ABB RobotStudio station: FinalSystem_Mark5.rspag

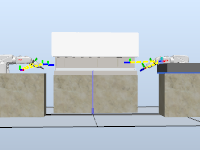
--- station ---
Station FinalSystem_Mark5 (saved by RobotStudio 20.1.8982.0)
Controller Brazo_Izquierdo, task T_ROB1: task frame (RAPID world) sits at (381.13, 1073.42, 0) mm, rotated rx 0 ry 0.08 rz -90.05 deg in the station
Controller Brazo_Derecho, task T_ROB1: task frame (RAPID world) sits at (383.2, -1129.52, 0) mm, rotated rx 0 ry 0 rz 90 deg in the station
Controller Brazo_Derecho
  mechanical unit ROB_1: Brazo_Derecho, 6 joints, base frame (0, 0, 0) mm
Controller Brazo_Izquierdo
  mechanical unit ROB_1: Brazo_Izquierdo, 6 joints, base frame (0, 0, 0) mm
Layout (positions relative to the parent item):
  - Drunk machine [part] at (-616.69, -0.57, 747.91) mm, rotated rx 90.16 ry 0 rz 90.05 deg
  - rack [part] at (-166.71, -1080.65, 472.06) mm
  - ASS Nastro 80 [graphiccomponentgroup] at (220.02, -32.24, 435.23) mm, rotated rx -89.85 ry 0 rz 90.13 deg
    - Spalla ant tappeto-1 [part] at (3.95, -82.87, -3) mm
    - Tappeto L500 d80-1 [part] at (-9.66, -82.87, -105) mm
    - Spalla post tappeto 80-2 [part] at (3.95, -82.87, -207) mm
    - Traversa supporto piano di lavoro Nastro 80-1 [part] at (3.95, -77.67, -105) mm
    - Traversa supporto piano di lavoro Nastro 80-2 [part] at (363.95, -77.67, -105) mm
    - Traversa supporto piano di lavoro Nastro 80-3 [part] at (243.95, -77.67, -105) mm
    - Traversa supporto piano di lavoro Nastro 80-4 [part] at (123.95, -77.67, -105) mm
    - Traversa supporto piano di lavoro Nastro 80-5 [part] at (-116.05, -77.67, -105) mm
    - Ass rullo passivo Nastro 80-1 [graphiccomponentgroup] at (-483.55, -82.94, -125) mm, rotated rx 0 ry 0 rz 115.98 deg
      - Albero rullo passivo 80-1 [part] at (-0.06, -0.28, -82) mm
      - Rullo passivo Nastro 80-1 [part] at (-0.06, -0.28, 20) mm, rotated rx 0 ry 0 rz 44.34 deg
      - Cuscinetto 6205-2RS1-2 [part] at (-0.06, -0.28, 121) mm, rotated rx 0 ry 90 rz -50.21 deg
      - Cuscinetto 6205-2RS1-3 [part] at (-0.06, -0.28, -75) mm, rotated rx 0 ry 90 rz -77.93 deg
    - Traversa supporto piano di lavoro Nastro 80-6 [part] at (-236.05, -77.67, -105) mm
    - Traversa supporto piano di lavoro Nastro 80-7 [part] at (-356.05, -77.67, -105) mm
    - Testa spalla front Nastro 80-1 [part] at (-483.27, -82.87, 0) mm
    - Testa spalla post Nastro 80-1 [part] at (-483.27, -82.87, -210) mm
  - Brazo_Izquierdo [mechanism, from Robots\IRB120_3_58_G_01.rslib] at (381.13, 1073.42, 0) mm, rotated rx 0 ry 0.08 rz -90.05 deg; joint values [0, 0, 0, 0, 0.5236, 1.5708] (rad or m)
  - Smart_Gripper_Servo_Fingers [mechanism, from Libraries\Smart_Gripper2.rslib] at (383.22, -765.16, 594) mm, rotated rx 120 ry 0 rz 180 deg; joint values [0.025] (rad or m)
  - Brazo_Derecho [mechanism, from Robots\IRB120_3_58_G_01.rslib] at (383.2, -1129.52, 0) mm, rotated rx 0 ry 0 rz 90 deg; joint values [0, 0, 0, 0, 0.5236, 1.5708] (rad or m)
  - Smart_Gripper_Servo_Fingers_2 [mechanism, from Tools\ABB_Smart_Gripper_Servo_Fingers.rslib] at (380.83, 708.25, 593.49) mm, rotated rx 120.08 ry 0 rz -0.05 deg; joint values [0.0241] (rad or m)
  - Base [part] at (176.64, -543.05, 0) mm
  - Vaso [part] at (55.85, -802.14, 590.8) mm
  - Positioner [smart component, from Components\Positioner.rslib]
      properties: Object=Vaso; Position=[0.055849 -0.80214 0.5908]; Orientation=[0 0 0]; Reference=Global; ReferenceObject=(none)
  - Sensor_Final [smart component, from Components\PlaneSensor.rslib] at (317.79, 437.34, 555.44) mm, rotated rx 90 ry 0 rz 0 deg
      properties: Origin=[0 0 0]; Axis1=[0.1 0 0]; Axis2=[0 0.1 0]; SensedPart=(none)
    - _sensorPart_ [part, from Components\PlaneSensor.rslib]
  - SimulationEvents [smart component, from Components\SimulationEvents.rslib]
  - LogicSRLatch [smart component, from Components\LogicSRLatch.rslib]
  - LinearMover_I-H [smart component, from Components\LinearMover.rslib]
      properties: Object=Vaso; Direction=[0 0.1 0]; Speed=0.06; Reference=Global; ReferenceObject=(none)
  - Detacher [smart component, from Components\Detacher.rslib]
      properties: Child=Vaso; KeepPosition=true
  - Sensor_Hielos [smart component, from Components\PlaneSensor.rslib] at (291.31, -320.38, 553.19) mm, rotated rx 90 ry 0 rz 0 deg
      properties: Origin=[0 0 0]; Axis1=[0.1 0 0]; Axis2=[0 0.1 0]; SensedPart=(none)
    - _sensorPart_ [part, from Components\PlaneSensor.rslib]
  - Attacher_2 [smart component, from Components\Attacher.rslib]
      properties: Parent=Smart_Gripper_Servo_Fingers_2; Flange=0; Child=Vaso; Mount=false; Offset=[0 0 0]; Orientation=[0 0 0]
  - Pieza_8 [part] at (-304.73, -1255.96, -1.15) mm
  - Pieza_9 [part] at (-221.9, 531.96, -0.59) mm
  - Attacher_3 [smart component, from Components\Attacher.rslib]
      properties: Parent=Smart_Gripper_Servo_Fingers; Flange=0; Child=Vaso; Mount=false; Offset=[0 0 0]; Orientation=[0 0 0]
  - Detacher_2 [smart component, from Components\Detacher.rslib]
      properties: Child=Vaso; KeepPosition=true
  - LinearMover_H-A [smart component, from Components\LinearMover.rslib]
      properties: Object=Vaso; Direction=[0 0.1 0]; Speed=0.06; Reference=Global; ReferenceObject=(none)
  - LogicSRLatch_2 [smart component, from Components\LogicSRLatch.rslib]
  - Sensor_Tequila [smart component, from Components\PlaneSensor.rslib] at (290.86, -66.85, 550.9) mm, rotated rx 90 ry 0 rz 0 deg
      properties: Origin=[0 0 0]; Axis1=[0.1 0 0]; Axis2=[0 0.1 0]; SensedPart=(none)
    - _sensorPart_ [part, from Components\PlaneSensor.rslib]
  - LinearMover_A-M [smart component, from Components\LinearMover.rslib]
      properties: Object=Vaso; Direction=[0 0.1 0]; Speed=0.06; Reference=Global; ReferenceObject=(none)
  - LogicSRLatch_3 [smart component, from Components\LogicSRLatch.rslib]
  - Sensor_Toronja [smart component, from Components\PlaneSensor.rslib] at (305.49, 235.87, 549.38) mm, rotated rx 90 ry 0 rz 0 deg
      properties: Origin=[0 0 0]; Axis1=[0.1 0 0]; Axis2=[0 0.1 0]; SensedPart=(none)
    - _sensorPart_ [part, from Components\PlaneSensor.rslib]
  - LogicSRLatch_4 [smart component, from Components\LogicSRLatch.rslib]
  - LinearMover_M-F [smart component, from Components\LinearMover.rslib]
      properties: Object=Vaso; Direction=[0 0.1 0]; Speed=0.06; Reference=Global; ReferenceObject=(none)
  - Sensor_Coca [smart component, from Components\PlaneSensor.rslib] at (296.45, 334.57, 549.82) mm, rotated rx 90 ry 0 rz 0 deg
      properties: Origin=[0 0 0]; Axis1=[0.1 0 0]; Axis2=[0 0.1 0]; SensedPart=(none)
    - _sensorPart_ [part, from Components\PlaneSensor.rslib]
  - LogicSRLatch_5 [smart component, from Components\LogicSRLatch.rslib]
  - Sensor_Sprite [smart component, from Components\PlaneSensor.rslib] at (304.78, 430.43, 554.72) mm, rotated rx 90 ry 0 rz 0 deg
      properties: Origin=[0 0 0]; Axis1=[0.1 0 0]; Axis2=[0 0.1 0]; SensedPart=(none)
    - _sensorPart_ [part, from Components\PlaneSensor.rslib]
  - LogicSRLatch_6 [smart component, from Components\LogicSRLatch.rslib]
  - LogicSRLatch_7 [smart component, from Components\LogicSRLatch.rslib]
  - Sensor_Vodka [smart component, from Components\PlaneSensor.rslib] at (307.92, 135.66, 549.24) mm, rotated rx 90 ry 0 rz 0 deg
      properties: Origin=[0 0 0]; Axis1=[0.1 0 0]; Axis2=[0 0.1 0]; SensedPart=(none)
    - _sensorPart_ [part, from Components\PlaneSensor.rslib]
Attachment: Smart_Gripper_Servo_Fingers is attached to Brazo_Derecho / Link6
Attachment: Smart_Gripper_Servo_Fingers_2 is attached to Brazo_Izquierdo / Link6
Station signals: DI Posicionador
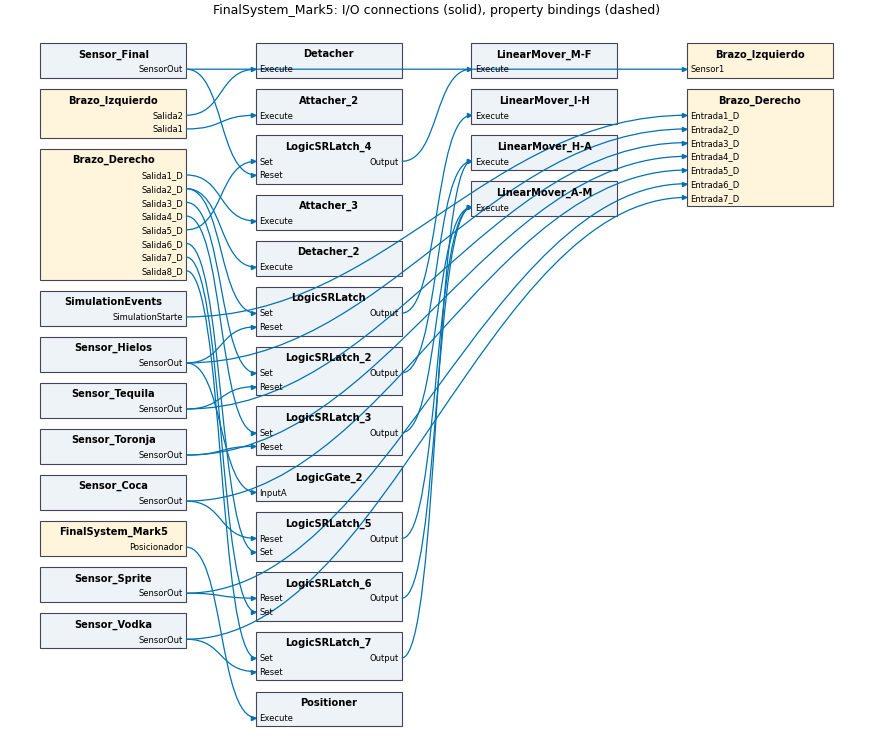
Station logic (signal -> signal, property => property):
  Sensor_Final.SensorOut -> Brazo_Izquierdo.Sensor1
  LogicSRLatch.Output -> LinearMover_I-H.Execute
  Brazo_Izquierdo.Salida2 -> Detacher.Execute
  Brazo_Izquierdo.Salida1 -> Attacher_2.Execute
  Brazo_Derecho.Salida1_D -> Attacher_3.Execute
  Brazo_Derecho.Salida2_D -> Detacher_2.Execute
  SimulationEvents.SimulationStarted -> Brazo_Derecho.Entrada1_D
  Sensor_Hielos.SensorOut -> LogicGate_2.InputA
  Brazo_Derecho.Salida2_D -> LogicSRLatch.Set
  Sensor_Hielos.SensorOut -> LogicSRLatch.Reset
  Brazo_Derecho.Salida3_D -> LogicSRLatch_2.Set
  LogicSRLatch_2.Output -> LinearMover_H-A.Execute
  Sensor_Hielos.SensorOut -> Brazo_Derecho.Entrada2_D
  Brazo_Derecho.Salida4_D -> LogicSRLatch_3.Set
  LogicSRLatch_3.Output -> LinearMover_A-M.Execute
  Sensor_Tequila.SensorOut -> Brazo_Derecho.Entrada3_D
  Sensor_Tequila.SensorOut -> LogicSRLatch_2.Reset
  Sensor_Toronja.SensorOut -> Brazo_Derecho.Entrada4_D
  Sensor_Toronja.SensorOut -> LogicSRLatch_3.Reset
  Brazo_Derecho.Salida5_D -> LogicSRLatch_4.Set
  Sensor_Final.SensorOut -> LogicSRLatch_4.Reset
  LogicSRLatch_4.Output -> LinearMover_M-F.Execute
  Sensor_Coca.SensorOut -> Brazo_Derecho.Entrada5_D
  FinalSystem_Mark5.Posicionador -> Positioner.Execute
  LogicSRLatch_5.Output -> LinearMover_A-M.Execute
  Sensor_Coca.SensorOut -> LogicSRLatch_5.Reset
  Brazo_Derecho.Salida6_D -> LogicSRLatch_5.Set
  Sensor_Sprite.SensorOut -> Brazo_Derecho.Entrada6_D
  Sensor_Sprite.SensorOut -> LogicSRLatch_6.Reset
  Brazo_Derecho.Salida7_D -> LogicSRLatch_6.Set
  LogicSRLatch_6.Output -> LinearMover_A-M.Execute
  Sensor_Vodka.SensorOut -> Brazo_Derecho.Entrada7_D
  Brazo_Derecho.Salida8_D -> LogicSRLatch_7.Set
  Sensor_Vodka.SensorOut -> LogicSRLatch_7.Reset
  LogicSRLatch_7.Output -> LinearMover_H-A.Execute

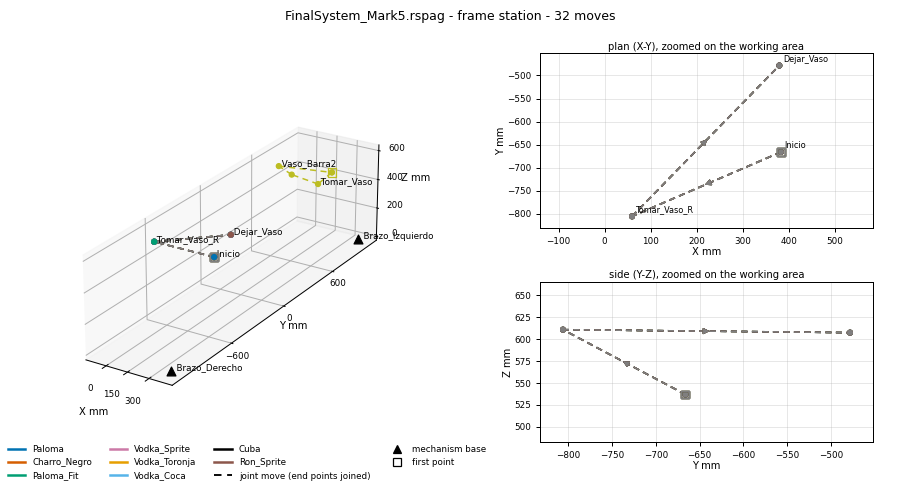
[picture p0: tool path of FinalSystem_Mark5.rspag in frame station, 32 of 32 moves have a stored position in this frame; points joined in program order, loops and branches not executed]
--- Backups/Brazo_Derecho/RAPID/TASK1/PROGMOD/CalibData.mod ---
MODULE CalibData
    PERS tooldata Servo:=[TRUE,[[0,0,114.2],[1,0,0,0]],[0.215,[8.7,12.3,49.2],[1,0,0,0],0.00021,0.00024,0.00009]];
ENDMODULE

--- Backups/Brazo_Derecho/RAPID/TASK1/PROGMOD/Module1.mod ---
MODULE Module1
    CONST robtarget Home:=[[463.253923278,0,536.899988039],[0.353553368,0.612372449,0.612372449,0.353553368],[0,-1,1,0],[9E+09,9E+09,9E+09,9E+09,9E+09,9E+09]];
    CONST robtarget AbovePickPosition:=[[323.968763837,312.895755919,276.594],[0.707106781,-0.707106781,-0.000020041,0.000020041],[0,0,0,0],[9E+09,9E+09,9E+09,9E+09,9E+09,9E+09]];
    CONST robtarget PickPosition:=[[323.968763837,312.895755919,156.594],[0.707106781,-0.707106781,-0.000020041,0.000020041],[0,0,0,0],[9E+09,9E+09,9E+09,9E+09,9E+09,9E+09]];
    CONST robtarget Inicio:=[[463.253923278,0,536.899988039],[0.353553368,0.612372449,0.612372449,0.353553368],[0,-1,1,0],[9E+09,9E+09,9E+09,9E+09,9E+09,9E+09]];
    CONST robtarget Tomar_Vaso_R:=[[323.459576854,323.459552433,610.906782794],[0.265834211,0.275279486,0.664583392,0.641780564],[0,0,1,0],[9E+09,9E+09,9E+09,9E+09,9E+09,9E+09]];
    CONST robtarget Dejar_Vaso:=[[651.164684644,3.54793506,607.492960443],[0.494318369,0.503022234,0.50566295,0.496913436],[0,-1,1,0],[9E+09,9E+09,9E+09,9E+09,9E+09,9E+09]];
   PROC main()
!        VAR socketdev server_socket;
!        VAR socketdev client_socket;
!        VAR string client_ip;
!        VAR string drinkID;
!        VAR bool loop:=TRUE;


!        SocketCreate server_socket;
!        SocketBind server_socket, "127.0.0.1", 55555;
!        SocketListen server_socket;

        ! Waiting for a connection request
!        SocketAccept server_socket, client_socket\ClientAddress:=client_ip\Time:=WAIT_MAX;

!        WHILE loop DO

!            SocketReceive client_socket \Str := drinkID\Time:=WAIT_MAX;

            !State machine
!            IF drinkID="id" THEN
!                !Mover izquierda
!                TPWrite "Izquierda";
!                Path_10;
!            ENDIF

!            drinkID := "";

            !Send acknowledge
            !SocketSend client_socket \Str := "Hello client with ip-addres " +client_ip;
!        ENDWHILE
!    ERROR
!        RETRY;
!    UNDO
!        SocketClose server_socket;
!        SocketClose client_socket;
        !Paloma;
        !Charro_Negro;
        !Paloma_Fit;
        !Vodka_Sprite;
        !Vodka_Toronja;
        !Vodka_Coca;
        !Cuba;
        !Ron_Sprite;
        Ron_Toronja;
    ENDPROC

    PROC Paloma()
        SetDO Salida1_D,0;
        SetDO Salida2_D,0;
        SetDO Salida3_D,0;
        SetDO Salida4_D,0;
        SetDO Salida5_D,0;
        SetDO Salida6_D,0;
        SetDO Salida7_D,0;
        SetDO Salida8_D,0;
        SetDO Salida9_D,0;

        !Movimiento Inicial Secuencia
        WaitDI Entrada1_D,1; !Espera a que se inicie la simulación
        MoveJ Inicio,v100,fine,Servo\WObj:=wobj0;!Mueve el brazo a posicion Inicial
        WaitTime 1;!Espera un segundo
        MoveJ Tomar_Vaso_R,v1000,fine,Servo\WObj:=wobj0;!Mueve el brazo a tomar el vaso
        WaitTime 1;!Espera un segundo
        SetDO Salida1_D,1;!Inicializa la salida1 a 1 para atach el vaso
        WaitTime 1;!Espera un segundo
        MoveJ Dejar_Vaso,v1000,fine,Servo\WObj:=wobj0; !Mueve el brazo y el vaso a la conveyor belt
        WaitTime 1;!Espera un segundo
        SetDO Salida1_D,0;!Inicializa la salida1 a 0 para deatach el vaso

        !Movimiento de Inicio a Sensor Hielos
        SetDO Salida2_D,1;!Inicializa la salida2 a 1 para iniciar LinearMover_I-H
        WaitTime 1;!Espera un segundo
        SetDO Salida2_D,0;!Inicializa la salida2 a 0 para evitar inicializar el LinearMover_I-H de nuevo.
        WaitDI Entrada2_D,1;!Espera a que el sensor hielos se active y para el movimiento.
        WaitTime 3;!Espera tres segundos en servir hielos

        !Movimiento de Sensor Hielos a Sensor A1
        SetDO Salida3_D,1;!Inicializa la salida3 a 1 para iniciar LinearMover_H-A
        WaitTime 1;!Espera un segundo
        SetDO Salida3_D,0;!Inicializa la salida3 a 0 para evitar inicializar el LinearMover_I-H de nuevo.
        WaitDI Entrada3_D,1;
        WaitTime 4;!Espera cuatro segundos en servir alcohol

        !Movimiento de Sensor A1 a Sensor M1
        SetDO Salida4_D,1;!Inicializa la salida4 a 1 para iniciar LinearMover_A-M
        WaitTime 1;!Espera un segundo
        SetDO Salida4_D,0;!Inicializa la salida4 a 0 para evitar inicializar el LinearMover_I-H de nuevo.
        WaitDI Entrada4_D,1;
        WaitTime 7;!Espera siete segundos en servir mixer

        !Movimiento de Sensor M1 a Sensor Final
        SetDO Salida5_D,1; !Inicializa la salida5 a 1 para iniciar LinearMover_M-F
        WaitTime 1;!Espera un segundo
        SetDO Salida5_D,0;!Inicializa la salida4 a 0 para evitar inicializar el LinearMover_I-H de nuevo.
    ENDPROC

    PROC Charro_Negro()
        SetDO Salida1_D,0;
        SetDO Salida2_D,0;
        SetDO Salida3_D,0;
        SetDO Salida4_D,0;
        SetDO Salida5_D,0;
        SetDO Salida6_D,0;
        SetDO Salida7_D,0;
        SetDO Salida8_D,0;
        SetDO Salida9_D,0;

        !Movimiento Inicial Secuencia
        WaitDI Entrada1_D,1; !Espera a que se inicie la simulación
        MoveJ Inicio,v100,fine,Servo\WObj:=wobj0;!Mueve el brazo a posicion Inicial
        WaitTime 1;!Espera un segundo
        MoveJ Tomar_Vaso_R,v1000,fine,Servo\WObj:=wobj0;!Mueve el brazo a tomar el vaso
        WaitTime 1;!Espera un segundo
        SetDO Salida1_D,1;!Inicializa la salida1 a 1 para atach el vaso
        WaitTime 1;!Espera un segundo
        MoveJ Dejar_Vaso,v1000,fine,Servo\WObj:=wobj0; !Mueve el brazo y el vaso a la conveyor belt
        WaitTime 1;!Espera un segundo
        SetDO Salida1_D,0;!Inicializa la salida1 a 0 para deatach el vaso

        !Movimiento de Inicio a Sensor Hielos
        SetDO Salida2_D,1;!Inicializa la salida2 a 1 para iniciar LinearMover_I-H
        WaitTime 1;!Espera un segundo
        SetDO Salida2_D,0;!Inicializa la salida2 a 0 para evitar inicializar el LinearMover_I-H de nuevo.
        WaitDI Entrada2_D,1;!Espera a que el sensor hielos se active y para el movimiento.
        WaitTime 3;!Espera tres segundos en servir hielos

        !Movimiento de Sensor Hielos a Sensor Tequila
        SetDO Salida3_D,1;!Inicializa la salida3 a 1 para iniciar LinearMover_H-A
        WaitTime 1;!Espera un segundo
        SetDO Salida3_D,0;!Inicializa la salida3 a 0 para evitar inicializar el LinearMover_H-A de nuevo.
        WaitDI Entrada3_D,1;
        WaitTime 4;!Espera cuatro segundos en servir alcohol

        !Movimiento de Sensor Tequila a Sensor Coca
        SetDO Salida6_D,1;!Inicializa la salida7 a 1 para iniciar LinearMover_A-M
        WaitTime 1;!Espera un segundo
        SetDO Salida6_D,0;!Inicializa la salida4 a 0 para evitar inicializar el LinearMover_I-H de nuevo.
        WaitDI Entrada5_D,1;
        WaitTime 7;!Espera siete segundos en servir mixer

        !Movimiento de Sensor M1 a Sensor Final
        SetDO Salida5_D,1; !Inicializa la salida5 a 1 para iniciar LinearMover_M-F
        WaitTime 1;!Espera un segundo
        SetDO Salida5_D,0;!Inicializa la salida4 a 0 para evitar inicializar el LinearMover_I-H de nuevo.
    ENDPROC

    PROC Paloma_Fit()
        SetDO Salida1_D,0;
        SetDO Salida2_D,0;
        SetDO Salida3_D,0;
        SetDO Salida4_D,0;
        SetDO Salida5_D,0;
        SetDO Salida6_D,0;
        SetDO Salida7_D,0;
        SetDO Salida8_D,0;
        SetDO Salida9_D,0;

        !Movimiento Inicial Secuencia
        WaitDI Entrada1_D,1; !Espera a que se inicie la simulación
        MoveJ Inicio,v100,fine,Servo\WObj:=wobj0;!Mueve el brazo a posicion Inicial
        WaitTime 1;!Espera un segundo
        MoveJ Tomar_Vaso_R,v1000,fine,Servo\WObj:=wobj0;!Mueve el brazo a tomar el vaso
        WaitTime 1;!Espera un segundo
        SetDO Salida1_D,1;!Inicializa la salida1 a 1 para atach el vaso
        WaitTime 1;!Espera un segundo
        MoveJ Dejar_Vaso,v1000,fine,Servo\WObj:=wobj0; !Mueve el brazo y el vaso a la conveyor belt
        WaitTime 1;!Espera un segundo
        SetDO Salida1_D,0;!Inicializa la salida1 a 0 para deatach el vaso

        !Movimiento de Inicio a Sensor Hielos
        SetDO Salida2_D,1;!Inicializa la salida2 a 1 para iniciar LinearMover_I-H
        WaitTime 1;!Espera un segundo
        SetDO Salida2_D,0;!Inicializa la salida2 a 0 para evitar inicializar el LinearMover_I-H de nuevo.
        WaitDI Entrada2_D,1;!Espera a que el sensor hielos se active y para el movimiento.
        WaitTime 3;!Espera tres segundos en servir hielos

        !Movimiento de Sensor Hielos a Sensor Tequila
        SetDO Salida3_D,1;!Inicializa la salida3 a 1 para iniciar LinearMover_H-A
        WaitTime 1;!Espera un segundo
        SetDO Salida3_D,0;!Inicializa la salida3 a 0 para evitar inicializar el LinearMover_H-A de nuevo.
        WaitDI Entrada3_D,1;
        WaitTime 4;!Espera cuatro segundos en servir alcohol

        !Movimiento de Sensor Tequila a Sensor Sprite
        SetDO Salida7_D,1;!Inicializa la salida4 a 1 para iniciar LinearMover_A-M
        WaitTime 1;!Espera un segundo
        SetDO Salida7_D,0;!Inicializa la salida4 a 0 para evitar inicializar el LinearMover_I-H de nuevo.
        WaitDI Entrada6_D,1;
        WaitTime 7;!Espera siete segundos en servir mixer

        !Movimiento de Sensor M1 a Sensor Final/Sprite
        SetDO Salida5_D,1; !Inicializa la salida5 a 1 para iniciar LinearMover_M-F
        WaitTime 1;!Espera un segundo
        SetDO Salida5_D,0;!Inicializa la salida4 a 0 para evitar inicializar el LinearMover_I-H de nuevo.
    ENDPROC

    PROC Vodka_Sprite()
        SetDO Salida1_D,0;
        SetDO Salida2_D,0;
        SetDO Salida3_D,0;
        SetDO Salida4_D,0;
        SetDO Salida5_D,0;
        SetDO Salida6_D,0;
        SetDO Salida7_D,0;
        SetDO Salida8_D,0;
        SetDO Salida9_D,0;

        !Movimiento Inicial Secuencia
        WaitDI Entrada1_D,1; !Espera a que se inicie la simulación
        MoveJ Inicio,v100,fine,Servo\WObj:=wobj0;!Mueve el brazo a posicion Inicial
        WaitTime 1;!Espera un segundo
        MoveJ Tomar_Vaso_R,v1000,fine,Servo\WObj:=wobj0;!Mueve el brazo a tomar el vaso
        WaitTime 1;!Espera un segundo
        SetDO Salida1_D,1;!Inicializa la salida1 a 1 para atach el vaso
        WaitTime 1;!Espera un segundo
        MoveJ Dejar_Vaso,v1000,fine,Servo\WObj:=wobj0; !Mueve el brazo y el vaso a la conveyor belt
        WaitTime 1;!Espera un segundo
        SetDO Salida1_D,0;!Inicializa la salida1 a 0 para deatach el vaso

        !Movimiento de Inicio a Sensor Hielos
        SetDO Salida2_D,1;!Inicializa la salida2 a 1 para iniciar LinearMover_I-H
        WaitTime 1;!Espera un segundo
        SetDO Salida2_D,0;!Inicializa la salida2 a 0 para evitar inicializar el LinearMover_I-H de nuevo.
        WaitDI Entrada2_D,1;!Espera a que el sensor hielos se active y para el movimiento.
        WaitTime 3;!Espera tres segundos en servir hielos

        !Movimiento de Sensor Hielos a Sensor Vodka
        SetDO Salida8_D,1;!Inicializa la salida3 a 1 para iniciar LinearMover_H-A
        WaitTime 1;!Espera un segundo
        SetDO Salida8_D,0;!Inicializa la salida3 a 0 para evitar inicializar el LinearMover_H-A de nuevo.
        WaitDI Entrada7_D,1;
        WaitTime 4;!Espera cuatro segundos en servir alcohol

        !Movimiento de Sensor Vodka a Sensor Sprite
        SetDO Salida7_D,1;!Inicializa la salida4 a 1 para iniciar LinearMover_A-M
        WaitTime 1;!Espera un segundo
        SetDO Salida7_D,0;!Inicializa la salida4 a 0 para evitar inicializar el LinearMover_I-H de nuevo.
        WaitDI Entrada6_D,1;
        WaitTime 7;!Espera siete segundos en servir mixer

        !Movimiento de Sensor M1 a Sensor Final/Sprite
        SetDO Salida5_D,1; !Inicializa la salida5 a 1 para iniciar LinearMover_M-F
        WaitTime 1;!Espera un segundo
        SetDO Salida5_D,0;!Inicializa la salida4 a 0 para evitar inicializar el LinearMover_I-H de nuevo.
    ENDPROC

    PROC Vodka_Toronja()
        SetDO Salida1_D,0;
        SetDO Salida2_D,0;
        SetDO Salida3_D,0;
        SetDO Salida4_D,0;
        SetDO Salida5_D,0;
        SetDO Salida6_D,0;
        SetDO Salida7_D,0;
        SetDO Salida8_D,0;
        SetDO Salida9_D,0;

        !Movimiento Inicial Secuencia
        WaitDI Entrada1_D,1; !Espera a que se inicie la simulación
        MoveJ Inicio,v100,fine,Servo\WObj:=wobj0;!Mueve el brazo a posicion Inicial
        WaitTime 1;!Espera un segundo
        MoveJ Tomar_Vaso_R,v1000,fine,Servo\WObj:=wobj0;!Mueve el brazo a tomar el vaso
        WaitTime 1;!Espera un segundo
        SetDO Salida1_D,1;!Inicializa la salida1 a 1 para atach el vaso
        WaitTime 1;!Espera un segundo
        MoveJ Dejar_Vaso,v1000,fine,Servo\WObj:=wobj0; !Mueve el brazo y el vaso a la conveyor belt
        WaitTime 1;!Espera un segundo
        SetDO Salida1_D,0;!Inicializa la salida1 a 0 para deatach el vaso

        !Movimiento de Inicio a Sensor Hielos
        SetDO Salida2_D,1;!Inicializa la salida2 a 1 para iniciar LinearMover_I-H
        WaitTime 1;!Espera un segundo
        SetDO Salida2_D,0;!Inicializa la salida2 a 0 para evitar inicializar el LinearMover_I-H de nuevo.
        WaitDI Entrada2_D,1;!Espera a que el sensor hielos se active y para el movimiento.
        WaitTime 3;!Espera tres segundos en servir hielos

        !Movimiento de Sensor Hielos a Sensor Vodka
        SetDO Salida8_D,1;!Inicializa la salida3 a 1 para iniciar LinearMover_H-A
        WaitTime 1;!Espera un segundo
        SetDO Salida8_D,0;!Inicializa la salida3 a 0 para evitar inicializar el LinearMover_H-A de nuevo.
        WaitDI Entrada7_D,1;
        WaitTime 4;!Espera cuatro segundos en servir alcohol

        !Movimiento de Sensor Vodka a Sensor Toronja
        SetDO Salida4_D,1;!Inicializa la salida4 a 1 para iniciar LinearMover_A-M
        WaitTime 1;!Espera un segundo
        SetDO Salida4_D,0;!Inicializa la salida4 a 0 para evitar inicializar el LinearMover_I-H de nuevo.
        WaitDI Entrada4_D,1;
        WaitTime 7;!Espera siete segundos en servir mixer

        !Movimiento de Sensor M1 a Sensor Final/Sprite
        SetDO Salida5_D,1; !Inicializa la salida5 a 1 para iniciar LinearMover_M-F
        WaitTime 1;!Espera un segundo
        SetDO Salida5_D,0;!Inicializa la salida4 a 0 para evitar inicializar el LinearMover_I-H de nuevo.
    ENDPROC

    PROC Vodka_Coca()
        SetDO Salida1_D,0;
        SetDO Salida2_D,0;
        SetDO Salida3_D,0;
        SetDO Salida4_D,0;
        SetDO Salida5_D,0;
        SetDO Salida6_D,0;
        SetDO Salida7_D,0;
        SetDO Salida8_D,0;
        SetDO Salida9_D,0;

        !Movimiento Inicial Secuencia
        WaitDI Entrada1_D,1; !Espera a que se inicie la simulación
        MoveJ Inicio,v100,fine,Servo\WObj:=wobj0;!Mueve el brazo a posicion Inicial
        WaitTime 1;!Espera un segundo
        MoveJ Tomar_Vaso_R,v1000,fine,Servo\WObj:=wobj0;!Mueve el brazo a tomar el vaso
        WaitTime 1;!Espera un segundo
        SetDO Salida1_D,1;!Inicializa la salida1 a 1 para atach el vaso
        WaitTime 1;!Espera un segundo
        MoveJ Dejar_Vaso,v1000,fine,Servo\WObj:=wobj0; !Mueve el brazo y el vaso a la conveyor belt
        WaitTime 1;!Espera un segundo
        SetDO Salida1_D,0;!Inicializa la salida1 a 0 para deatach el vaso

        !Movimiento de Inicio a Sensor Hielos
        SetDO Salida2_D,1;!Inicializa la salida2 a 1 para iniciar LinearMover_I-H
        WaitTime 1;!Espera un segundo
        SetDO Salida2_D,0;!Inicializa la salida2 a 0 para evitar inicializar el LinearMover_I-H de nuevo.
        WaitDI Entrada2_D,1;!Espera a que el sensor hielos se active y para el movimiento.
        WaitTime 3;!Espera tres segundos en servir hielos

        !Movimiento de Sensor Hielos a Sensor Vodka
        SetDO Salida8_D,1;!Inicializa la salida3 a 1 para iniciar LinearMover_H-A
        WaitTime 1;!Espera un segundo
        SetDO Salida8_D,0;!Inicializa la salida3 a 0 para evitar inicializar el LinearMover_H-A de nuevo.
        WaitDI Entrada7_D,1;
        WaitTime 4;!Espera cuatro segundos en servir alcohol

        !Movimiento de Sensor Vodka a Sensor Coca
        SetDO Salida6_D,1;!Inicializa la salida7 a 1 para iniciar LinearMover_A-M
        WaitTime 1;!Espera un segundo
        SetDO Salida6_D,0;!Inicializa la salida4 a 0 para evitar inicializar el LinearMover_I-H de nuevo.
        WaitDI Entrada5_D,1;
        WaitTime 7;!Espera siete segundos en servir mixer

        !Movimiento de Sensor M1 a Sensor Final/Sprite
        SetDO Salida5_D,1; !Inicializa la salida5 a 1 para iniciar LinearMover_M-F
        WaitTime 1;!Espera un segundo
        SetDO Salida5_D,0;!Inicializa la salida4 a 0 para evitar inicializar el LinearMover_I-H de nuevo.
    ENDPROC

    PROC Cuba()
        SetDO Salida1_D,0;
        SetDO Salida2_D,0;
        SetDO Salida3_D,0;
        SetDO Salida4_D,0;
        SetDO Salida5_D,0;
        SetDO Salida6_D,0;
        SetDO Salida7_D,0;
        SetDO Salida8_D,0;
        SetDO Salida9_D,0;

        !Movimiento Inicial Secuencia
        WaitDI Entrada1_D,1; !Espera a que se inicie la simulación
        MoveJ Inicio,v100,fine,Servo\WObj:=wobj0;!Mueve el brazo a posicion Inicial
        WaitTime 1;!Espera un segundo
        MoveJ Tomar_Vaso_R,v1000,fine,Servo\WObj:=wobj0;!Mueve el brazo a tomar el vaso
        WaitTime 1;!Espera un segundo
        SetDO Salida1_D,1;!Inicializa la salida1 a 1 para atach el vaso
        WaitTime 1;!Espera un segundo
        MoveJ Dejar_Vaso,v1000,fine,Servo\WObj:=wobj0; !Mueve el brazo y el vaso a la conveyor belt
        WaitTime 1;!Espera un segundo
        SetDO Salida1_D,0;!Inicializa la salida1 a 0 para deatach el vaso

        !Movimiento de Inicio a Sensor Hielos
        SetDO Salida2_D,1;!Inicializa la salida2 a 1 para iniciar LinearMover_I-H
        WaitTime 1;!Espera un segundo
        SetDO Salida2_D,0;!Inicializa la salida2 a 0 para evitar inicializar el LinearMover_I-H de nuevo.
        WaitDI Entrada2_D,1;!Espera a que el sensor hielos se active y para el movimiento.
        WaitTime 3;!Espera tres segundos en servir hielos

        !Movimiento de Sensor Hielos a Sensor Ron
        SetDO Salida9_D,1;!Inicializa la salida3 a 1 para iniciar LinearMover_H-A
        WaitTime 1;!Espera un segundo
        SetDO Salida9_D,0;!Inicializa la salida3 a 0 para evitar inicializar el LinearMover_H-A de nuevo.
        WaitDI Entrada8_D,1;
        WaitTime 4;!Espera cuatro segundos en servir alcohol

        !Movimiento de Sensor Ron a Sensor Coca
        SetDO Salida6_D,1;!Inicializa la salida7 a 1 para iniciar LinearMover_A-M
        WaitTime 1;!Espera un segundo
        SetDO Salida6_D,0;!Inicializa la salida4 a 0 para evitar inicializar el LinearMover_I-H de nuevo.
        WaitDI Entrada5_D,1;
        WaitTime 7;!Espera siete segundos en servir mixer

        !Movimiento de Sensor M1 a Sensor Final/Sprite
        SetDO Salida5_D,1; !Inicializa la salida5 a 1 para iniciar LinearMover_M-F
        WaitTime 1;!Espera un segundo
        SetDO Salida5_D,0;!Inicializa la salida4 a 0 para evitar inicializar el LinearMover_I-H de nuevo.
    ENDPROC

    PROC Ron_Sprite()
        SetDO Salida1_D,0;
        SetDO Salida2_D,0;
        SetDO Salida3_D,0;
        SetDO Salida4_D,0;
        SetDO Salida5_D,0;
        SetDO Salida6_D,0;
        SetDO Salida7_D,0;
        SetDO Salida8_D,0;
        SetDO Salida9_D,0;

        !Movimiento Inicial Secuencia
        WaitDI Entrada1_D,1; !Espera a que se inicie la simulación
        MoveJ Inicio,v100,fine,Servo\WObj:=wobj0;!Mueve el brazo a posicion Inicial
        WaitTime 1;!Espera un segundo
        MoveJ Tomar_Vaso_R,v1000,fine,Servo\WObj:=wobj0;!Mueve el brazo a tomar el vaso
        WaitTime 1;!Espera un segundo
        SetDO Salida1_D,1;!Inicializa la salida1 a 1 para atach el vaso
        WaitTime 1;!Espera un segundo
        MoveJ Dejar_Vaso,v1000,fine,Servo\WObj:=wobj0; !Mueve el brazo y el vaso a la conveyor belt
        WaitTime 1;!Espera un segundo
        SetDO Salida1_D,0;!Inicializa la salida1 a 0 para deatach el vaso

        !Movimiento de Inicio a Sensor Hielos
        SetDO Salida2_D,1;!Inicializa la salida2 a 1 para iniciar LinearMover_I-H
        WaitTime 1;!Espera un segundo
        SetDO Salida2_D,0;!Inicializa la salida2 a 0 para evitar inicializar el LinearMover_I-H de nuevo.
        WaitDI Entrada2_D,1;!Espera a que el sensor hielos se active y para el movimiento.
        WaitTime 3;!Espera tres segundos en servir hielos

        !Movimiento de Sensor Hielos a Sensor Ron
        SetDO Salida9_D,1;!Inicializa la salida3 a 1 para iniciar LinearMover_H-A
        WaitTime 1;!Espera un segundo
        SetDO Salida9_D,0;!Inicializa la salida3 a 0 para evitar inicializar el LinearMover_H-A de nuevo.
        WaitDI Entrada8_D,1;
        WaitTime 4;!Espera cuatro segundos en servir alcohol

        !Movimiento de Sensor Ron a Sensor Sprite
        SetDO Salida7_D,1;!Inicializa la salida4 a 1 para iniciar LinearMover_A-M
        WaitTime 1;!Espera un segundo
        SetDO Salida7_D,0;!Inicializa la salida4 a 0 para evitar inicializar el LinearMover_I-H de nuevo.
        WaitDI Entrada6_D,1;
        WaitTime 7;!Espera siete segundos en servir mixer

        !Movimiento de Sensor M1 a Sensor Final/Sprite
        SetDO Salida5_D,1; !Inicializa la salida5 a 1 para iniciar LinearMover_M-F
        WaitTime 1;!Espera un segundo
        SetDO Salida5_D,0;!Inicializa la salida4 a 0 para evitar inicializar el LinearMover_I-H de nuevo.
    ENDPROC

    PROC Ron_Toronja()
        SetDO Salida1_D,0;
        SetDO Salida2_D,0;
        SetDO Salida3_D,0;
        SetDO Salida4_D,0;
        SetDO Salida5_D,0;
        SetDO Salida6_D,0;
        SetDO Salida7_D,0;
        SetDO Salida8_D,0;
        SetDO Salida9_D,0;

        !Movimiento Inicial Secuencia
        WaitDI Entrada1_D,1; !Espera a que se inicie la simulación
        MoveJ Inicio,v100,fine,Servo\WObj:=wobj0;!Mueve el brazo a posicion Inicial
        WaitTime 1;!Espera un segundo
        MoveJ Tomar_Vaso_R,v1000,fine,Servo\WObj:=wobj0;!Mueve el brazo a tomar el vaso
        WaitTime 1;!Espera un segundo
        SetDO Salida1_D,1;!Inicializa la salida1 a 1 para atach el vaso
        WaitTime 1;!Espera un segundo
        MoveJ Dejar_Vaso,v1000,fine,Servo\WObj:=wobj0; !Mueve el brazo y el vaso a la conveyor belt
        WaitTime 1;!Espera un segundo
        SetDO Salida1_D,0;!Inicializa la salida1 a 0 para deatach el vaso

        !Movimiento de Inicio a Sensor Hielos
        SetDO Salida2_D,1;!Inicializa la salida2 a 1 para iniciar LinearMover_I-H
        WaitTime 1;!Espera un segundo
        SetDO Salida2_D,0;!Inicializa la salida2 a 0 para evitar inicializar el LinearMover_I-H de nuevo.
        WaitDI Entrada2_D,1;!Espera a que el sensor hielos se active y para el movimiento.
        WaitTime 3;!Espera tres segundos en servir hielos

        !Movimiento de Sensor Hielos a Sensor Ron
        SetDO Salida9_D,1;!Inicializa la salida3 a 1 para iniciar LinearMover_H-A
        WaitTime 1;!Espera un segundo
        SetDO Salida9_D,0;!Inicializa la salida3 a 0 para evitar inicializar el LinearMover_H-A de nuevo.
        WaitDI Entrada8_D,1;
        WaitTime 4;!Espera cuatro segundos en servir alcohol

        !Movimiento de Sensor Ron a Sensor Sprite
        SetDO Salida4_D,1;!Inicializa la salida4 a 1 para iniciar LinearMover_A-M
        WaitTime 1;!Espera un segundo
        SetDO Salida4_D,0;!Inicializa la salida4 a 0 para evitar inicializar el LinearMover_I-H de nuevo.
        WaitDI Entrada4_D,1;
        WaitTime 7;!Espera siete segundos en servir mixer

        !Movimiento de Sensor M1 a Sensor Final/Sprite
        SetDO Salida5_D,1; !Inicializa la salida5 a 1 para iniciar LinearMover_M-F
        WaitTime 1;!Espera un segundo
        SetDO Salida5_D,0;!Inicializa la salida4 a 0 para evitar inicializar el LinearMover_I-H de nuevo.
    ENDPROC

!    PROC Path_10()
!        MoveL Home,v100,fine,Servo\WObj:=wobj0;
!        MoveL AbovePickPosition,v100,fine,Servo\WObj:=wobj0;
!        MoveL PickPosition,v100,fine,Servo\WObj:=wobj0;
!        MoveL AbovePickPosition,v100,fine,Servo\WObj:=wobj0;
!        MoveL Home,v100,fine,Servo\WObj:=wobj0;
!    ENDPROC


ENDMODULE

--- Backups/Brazo_Izquierdo/RAPID/TASK1/PROGMOD/Module1.mod ---
MODULE Module1
        CONST robtarget Inicio:=[[364.353829072,0.000001062,594],[0.353553382,0.612372448,0.612372423,0.353553399],[0,-1,1,0],[9E+09,9E+09,9E+09,9E+09,9E+09,9E+09]];
    CONST robtarget Tomar_Vaso:=[[536.490074056,0.000001563,575.629108182],[0.499991499,0.500008499,0.500008479,0.499991523],[0,0,1,0],[9E+09,9E+09,9E+09,9E+09,9E+09,9E+09]];
    CONST robtarget Vaso_Barra1:=[[490.108064883,-218.210128446,575.631589757],[0.593029664,0.593029601,0.385118037,0.385117914],[-1,0,0,0],[9E+09,9E+09,9E+09,9E+09,9E+09,9E+09]];
    CONST robtarget Vaso_Barra2:=[[264.24731303,-448.60287155,506.737568503],[0.688134973,0.676228379,0.184361021,0.187607175],[-1,-1,1,1],[9E+09,9E+09,9E+09,9E+09,9E+09,9E+09]];
    PROC main()
        Path_10;
    ENDPROC
    PROC Path_10()
        setdo Salida1,0;
        setdo Salida2,0;
        Movej Inicio,v1000,z100,tool0\WObj:=wobj0;
        WaitDI Sensor1,1;
        WaitTime 1;
        Movej Tomar_Vaso,v1000,z100,tool0\WObj:=wobj0;
        WaitTime 1;
        setdo Salida1,1;
        WaitTime 1;
        Movej Vaso_Barra1,v1000,z100,tool0\WObj:=wobj0;
        Movej Vaso_Barra2,v1000,z100,tool0\WObj:=wobj0;
        WaitTime 1;
        SetDO Salida1,0;
        SetDO Salida2,1;
        WaitTime 1;
        Movej Inicio,v1000,z100,tool0\WObj:=wobj0;
        WaitDI Sensor2,1;




    ENDPROC
ENDMODULE

--- Backups/Brazo_Derecho/SYSPAR/EIO.cfg ---
EIO:CFG_1.0:6:1::
#
INDUSTRIAL_NETWORK:

      -Name "EtherNetIP" -Connection "Private Network"\
      -Label "EtherNet/IP Adapter Network"

      -Name "DeviceNet" -Label "DeviceNet Master/Slave Network" -Address "2"
#
DEVICENET_INTERNAL_DEVICE:

      -Name "DN_Internal_Device" -VendorName "ABB Robotics"\
      -ProductName "DeviceNet Internal Slave Device"
#
ETHERNETIP_INTERNAL_DEVICE:

      -Name "EN_Internal_Device" -VendorName "ABB Robotics"\
      -ProductName "EtherNet/IP Internal Adapter Device"
#
EIO_SIGNAL:

      -Name "Salida1_D" -SignalType "DO" -Device "DN_Internal_Device"\
      -DeviceMap "0"

      -Name "Salida2_D" -SignalType "DO" -Device "DN_Internal_Device"\
      -DeviceMap "1"

      -Name "Entrada1_D" -SignalType "DI" -Device "DN_Internal_Device"\
      -DeviceMap "2"

      -Name "Entrada2_D" -SignalType "DI" -Device "DN_Internal_Device"\
      -DeviceMap "3"

      -Name "Salida3_D" -SignalType "DO" -Device "DN_Internal_Device"\
      -DeviceMap "4"

      -Name "Entrada3_D" -SignalType "DI" -Device "DN_Internal_Device"\
      -DeviceMap "5"

      -Name "Salida4_D" -SignalType "DO" -Device "DN_Internal_Device"\
      -DeviceMap "6"

      -Name "Entrada4_D" -SignalType "DI" -Device "DN_Internal_Device"\
      -DeviceMap "7"

      -Name "Salida5_D" -SignalType "DO" -Device "DN_Internal_Device"\
      -DeviceMap "8"

      -Name "Entrada5_D" -SignalType "DI" -Device "DN_Internal_Device"\
      -DeviceMap "9"

      -Name "Salida6_D" -SignalType "DO" -Device "DN_Internal_Device"\
      -DeviceMap "10"

      -Name "Entrada6_D" -SignalType "DI" -Device "DN_Internal_Device"\
      -DeviceMap "11"

      -Name "Salida7_D" -SignalType "DO" -Device "DN_Internal_Device"\
      -DeviceMap "12"

      -Name "Entrada7_D" -SignalType "DI" -Device "DN_Internal_Device"\
      -DeviceMap "13"

      -Name "Salida8_D" -SignalType "DO" -Device "DN_Internal_Device"\
      -DeviceMap "14"

      -Name "Entrada8_D" -SignalType "DI" -Device "DN_Internal_Device"\
      -DeviceMap "15"

      -Name "Salida9_D" -SignalType "DO" -Device "DN_Internal_Device"\
      -DeviceMap "16"

--- Backups/Brazo_Izquierdo/SYSPAR/EIO.cfg ---
EIO:CFG_1.0:6:1::
#
INDUSTRIAL_NETWORK:

      -Name "EtherNetIP" -Connection "Private Network"\
      -Label "EtherNet/IP Adapter Network"

      -Name "DeviceNet" -Label "DeviceNet Master/Slave Network" -Address "2"
#
DEVICENET_INTERNAL_DEVICE:

      -Name "DN_Internal_Device" -VendorName "ABB Robotics"\
      -ProductName "DeviceNet Internal Slave Device"
#
ETHERNETIP_INTERNAL_DEVICE:

      -Name "EN_Internal_Device" -VendorName "ABB Robotics"\
      -ProductName "EtherNet/IP Internal Adapter Device"
#
EIO_SIGNAL:

      -Name "Sensor1" -SignalType "DI" -Device "DN_Internal_Device"\
      -DeviceMap "0"

      -Name "Salida1" -SignalType "DO" -Device "DN_Internal_Device"\
      -DeviceMap "1"

      -Name "Salida2" -SignalType "DO" -Device "DN_Internal_Device"\
      -DeviceMap "2"

      -Name "Sensor2" -SignalType "DI" -Device "DN_Internal_Device"\
      -DeviceMap "3"
